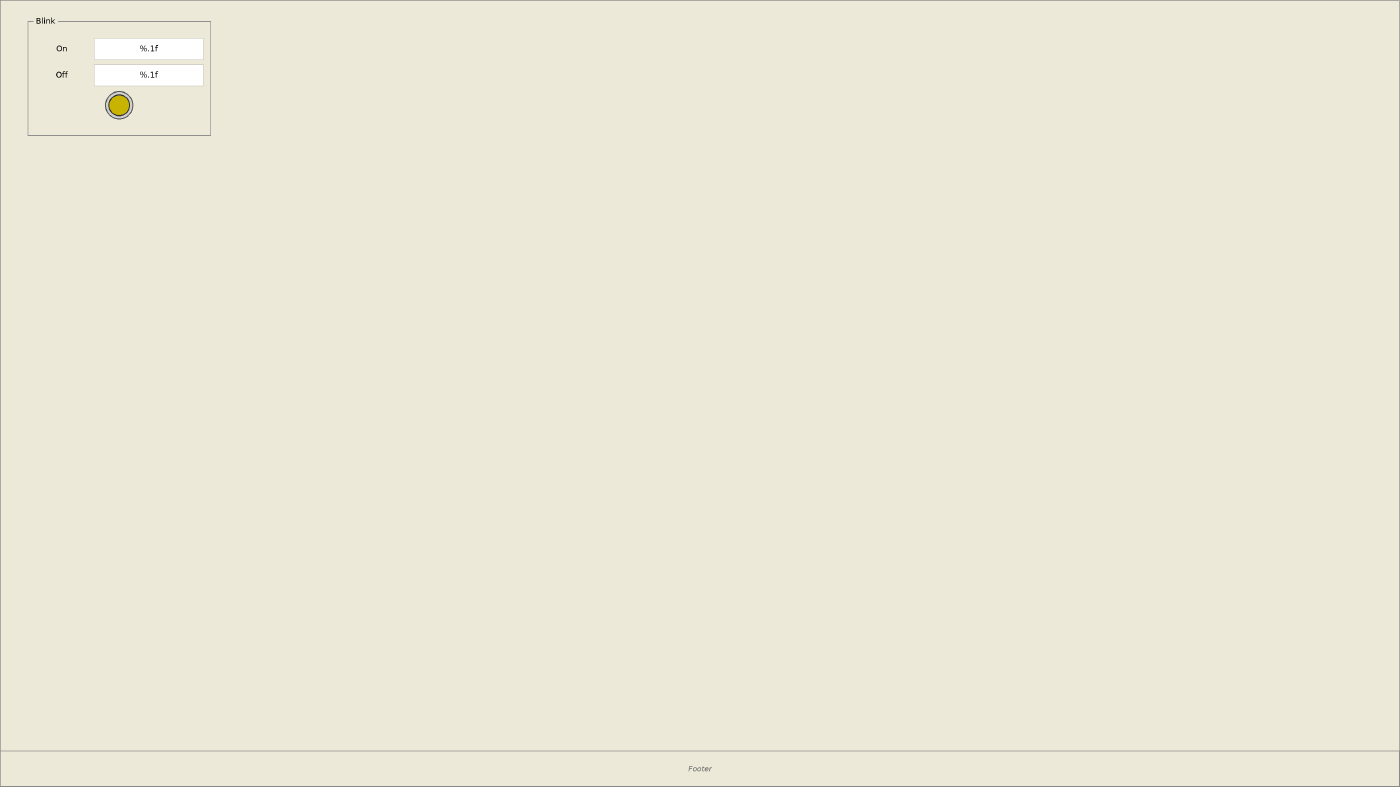
VISUALIZATION Visualization  // 1920x1080
    GroupBox (38,21 251x165), "Blink"
        Label (12,31 70x30), "On"
        Label (12,67 70x30), "Off"
        Lamp1 (103,101 45x45), variable: prgTestAuxsFuns.bOutputBlink, style: Lamp-Lamp1-Yellow
        Textfield (91,31 150x30), "%.1f", text variable: prgTestAuxsFuns.rBlinkOn
            OnMouseClick: write the text variable via Default
        Textfield (91,67 150x30), "%.1f", text variable: prgTestAuxsFuns.rBlinkOff
            OnMouseClick: write the text variable via Default
    Frame (0,1030 1920x50)
        shows Footer()
END_VISUALIZATION

(* stored: Version 1.1.0.1, ProductVersion 3.1.4024.12
   Visu Visualization: Id {17937c2f-499f-4307-a0b7-9b6eb0c5c429} *)
